{attribute 'linkalways'} 
{attribute 'no_explicit_call' := 'This FB is a CLASS and must be accessed using methods or properties'}
{attribute 'enable_dynamic_creation'}
FUNCTION_BLOCK FINAL NOT_INT EXTENDS Node
VAR
	in : _INT(0);
	out : _INT(0);
END_VAR

METHOD PUBLIC Clone : I_Node
VAR
	pNode : POINTER TO NOT_INT;
END_VAR
pNode := __NEW(NOT_INT);
Clone := pNode^;
END_METHOD

METHOD FB_init : BOOL
VAR_INPUT
	bInitRetains : BOOL; // if TRUE, the retain variables are initialized (warm start / cold start)
	bInCopyCode : BOOL;  // if TRUE, the instance afterwards gets moved into the copy code (online change)
END_VAR
AddInput('in',THIS^.in);
AddOutput('out', THIS^.out);
END_METHOD

METHOD PROTECTED OnExecute
VAR
END_VAR
out.Value := NOT in.Value;
END_METHOD

END_FUNCTION_BLOCK

(* stored: Version 1.1.0.1, ProductVersion 3.1.4024.15
   POU NOT_INT: Id {7e4d87fb-7c71-4703-b072-51c0ea0a4cf4}, SpecialFunc None
   Folder Constructor: Id {cfbf7cfb-7dd0-4432-b2a5-0c2aa3799324}
   Method Clone: Id {a1f07aec-74a0-4fcb-88fa-c1003b09632e}
   Method FB_init: Id {4b090f04-9b15-42ef-b6d0-245fcd87e8cb}
   Method OnExecute: Id {7ec5ba8f-2b8c-4100-a089-9a13f9915a1d} *)
